FUNCTION_BLOCK ABSTRACT TcoStateExtendible EXTENDS TcoStateBase

METHOD PROTECTED FINAL ChangeState : ITcoState
VAR_INPUT
	NewState : INT;
END_VAR
ChangeState := SUPER^.ChangeStateProtected(NewState);
END_METHOD

(*~
	<docu>
		<summary>
			This method is called on each change of the <c>State</c>. This method could be overloaded and custom code should be placed here.	
		</summary>			
	</docu>	
~*)
METHOD PROTECTED OnStateChange
VAR_INPUT
	PreviousState	: INT;
	NewState 		: INT;
END_VAR
SUPER^.OnStateChange(PreviousState, NewState);
END_METHOD

END_FUNCTION_BLOCK

(* stored: Version 1.1.0.1
   POU TcoStateExtendible: Id {0382c192-a9cc-0bc0-35e0-92f74a06fb79}, SpecialFunc None
   Method ChangeState: Id {bb1133c8-59fb-0b5a-0ba5-84fb713fd050}
   Method OnStateChange: Id {7e3711b4-64d6-0376-39cd-441141a47fe0} *)
